TYPE "UDT_Scl"
VERSION : 0.1
   STRUCT
      Count : Int;
   END_STRUCT;

END_TYPE
